{attribute 'qualified_only'}
{attribute 'strict'}
TYPE estadosHome :
(
	subiendo:=0,
	abriendo,
	sacando,
	ok,
	espera
);
END_TYPE

(* stored: Version 1.1.0.1, ProductVersion 3.1.4024.9
   DUT estadosHome: Id {c0aef8fc-121a-4e9d-9c12-1a11fbb2e05e} *)
